Staubli VAL3: ServerSend.pgx

public program ServerSend(string x_sMess (dimensions=1))
begin

  synServer=x_sMess


end
